Universal Robots PolyScope program: you.urp

Program you (installation=default directory=/programs/usbdisk createdIn=5.19.0 lastSavedIn=5.19.0 robotSerialNumber=20235366666)
Calibrated DH parameters: a=[-0.000074, -0.240481, -0.025105, 0.000089, -0.000025, 0]; d=[0.151722, 81.163768, -218.075848, 137.042846, 0.08536, 0.091978]; alpha=[1.570306, -0.000479, -0.001547, 1.572519, -1.572356, 0]; deltaTheta=[0, -0.16012, 1.612913, -1.452801, 0, 0]
InitVariablesNode
Robot Program (runOnlyOnce=false)
  MoveL speed 250 mm/s, acceleration 1200 mm/s^2 (useActiveTCP=true) feature=Base
    Waypoint Waypoint_1: TCP in base x=344.161 y=-83.486 z=466.172 mm, rx=0.0026 ry=-0.0197 rz=2.2489 rad; joints [-214.972, -2.242, -87.588, 0.188, 90.731, 73.914] deg
